// Mitsubishi GX Works2 project: INC_DEC 명령어   PLC: Q02/Q02H

PROGRAM MAIN
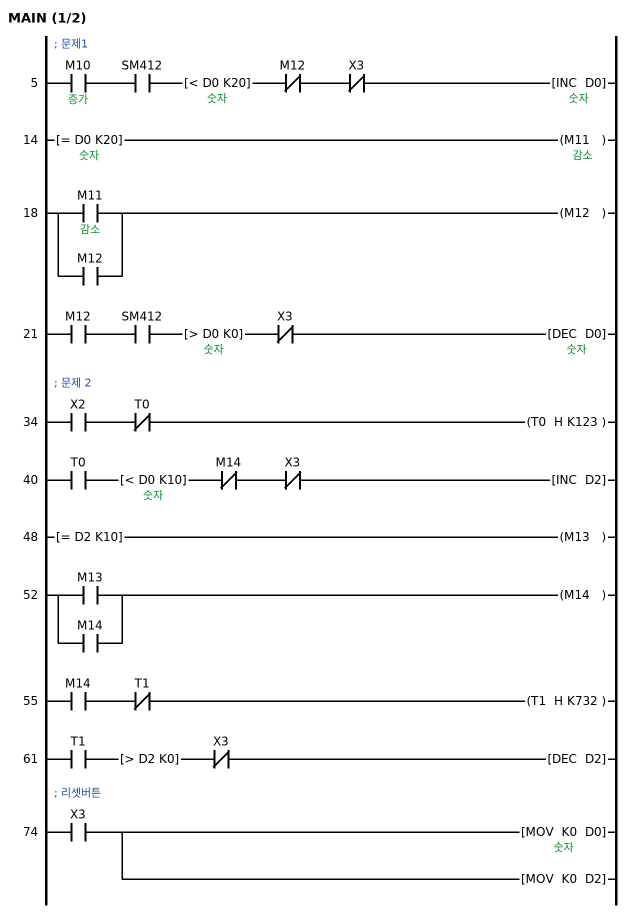
; 문제1
5     LD      M10  ; 증가
      AND     SM412
      AND<    D0 K20  ; 숫자
      ANI     M12
      ANI     X3
      INC     D0
14    LD=     D0 K20  ; 숫자
      OUT     M11  ; 감소
18    LD      M11  ; 감소
      OR      M12
      OUT     M12
21    LD      M12
      AND     SM412
      AND>    D0 K0  ; 숫자
      ANI     X3
      DEC     D0
; 문제 2
34    LD      X2
      ANI     T0
      OUTH    T0 K123
40    LD      T0
      AND<    D0 K10  ; 숫자
      ANI     M14
      ANI     X3
      INC     D2
48    LD=     D2 K10
      OUT     M13
52    LD      M13
      OR      M14
      OUT     M14
55    LD      M14
      ANI     T1
      OUTH    T1 K732
61    LD      T1
      AND>    D2 K0
      ANI     X3
      DEC     D2
; 리셋버튼
74    LD      X3
      MOV     K0 D0
      MOV     K0 D2
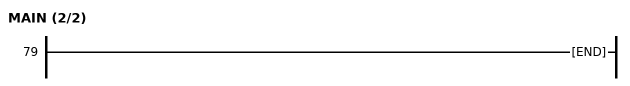
79    END
END_PROGRAM
